// TIA Portal V20 export
DATA_BLOCK "HMI_Interface_DeviceHistory"   // DB7
// stored: MemoryReserve 100
   VAR
      hotPressLeftHistory { ExternalWritable := 'False'; S7_SetPoint := 'True'} : "LER_typeVisionInspectData";
      hotPressRightHistory { ExternalWritable := 'False'; S7_SetPoint := 'True'} : "LER_typeVisionInspectData";
      hipotHistory { ExternalWritable := 'False'; S7_SetPoint := 'True'} : "LER_typeHipotDataLog";
      thicknessHistory { ExternalWritable := 'False'; S7_SetPoint := 'True'} : "LER_typeThicknessDataLog";
      visionHistory { ExternalWritable := 'False'; S7_SetPoint := 'True'} : "LER_typeVisionHistory";
      laserMarkHistory { ExternalWritable := 'False'; S7_SetPoint := 'True'} : "LER_typeQRMarkerDataLog";
      weightCheckHistory { ExternalWritable := 'False'; S7_SetPoint := 'True'} : "LER_typeWeightCheckDataLog";
   END_VAR
BEGIN
END_DATA_BLOCK
